TYPE LogGlobalArraySemStruct :
STRUCT
	//SemID : UDINT;
	//SemCreate_0 : SemCreate;
	//SemGetInfo_0 : SemGetInfo;
	SemaStat : UINT;
END_STRUCT
END_TYPE

(* stored: Version 1.1.0.1, ProductVersion 3.1.4024.3
   DUT LogGlobalArraySemStruct: Id {c66fb797-dd6e-0ab0-0e4c-d25b908e65b4} *)
